{attribute 'qualified_only'}
VAR_GLOBAL
    bGlobalTestFlag : BOOL;
END_VAR

(* stored: Version 1.1.0.1, ProductVersion 3.1.4024.12
   GVL GVL: Id {7ed94512-0cbc-4669-8f56-0baad7f9b2a2} *)
